TYPE T_SEC_ZXX7_ActiveExceptionStatus : USINT; END_TYPE

(* stored: Version 1.1.0.1, ProductVersion 3.1.4024.15
   DUT T_SEC_ZXX7_ActiveExceptionStatus: Id {da1c0cd7-cf39-0909-36f2-8b7c6e1ee254} *)
